Universal Robots PolyScope program: d_3.urp

Program d_3 (installation=ext_control directory=/programs createdIn=5.17.3 lastSavedIn=5.17.3 robotSerialNumber=20245501435)
Calibrated DH parameters: a=[0.000154, -0.137004, -0.385524, -0.00002, 0.000092, 0]; d=[0.162441, 211.794786, -230.585024, 18.923638, 0.099786, 0.09951]; alpha=[1.569493, -0.001902, 0.003874, 1.570111, -1.570167, 0]; deltaTheta=[0, -1.242934, 1.056292, 0.186646, 0.000002, 0.000001]
InitVariablesNode
Robot Program (runOnlyOnce=false)
  MoveL speed 250 mm/s, acceleration 1200 mm/s^2 (useActiveTCP=true) feature=Plane_2
    Waypoint Waypoint_1: TCP in base x=395.148 y=672.678 z=93.509 mm, rx=-1.4016 ry=-1.7845 rz=1.136 rad; joints [-134.118, -20.061, 52.844, -63.203, -64.354, -162.518] deg; TCP offset x=28.21 y=-96.107 z=-99.69 mm, rx=0 ry=0 rz=0 rad; feature pose in base x=343.605 y=747.803 z=100.778 mm, rx=2.6274 ry=0.0101 rz=1.3113 rad
    Waypoint Waypoint_2 (Relative): relativeFromPosition TCP in base x=395.142 y=672.688 z=93.545 mm, rx=-1.4016 ry=-1.7846 rz=1.136 rad; joints [-134.117, -20.063, 52.843, -63.203, -64.354, -162.518] deg; TCP in base x=394.531 y=580.607 z=100.773 mm, rx=-1.4016 ry=-1.7845 rz=1.1361 rad; joints [-139.249, -29.656, 72.902, -72.571, -68.776, -165.286] deg
